(*********************************** G.D S.p.A. - Technical Department ***********************************
============= PROGRAM INFO ============
FOLDER:             TBD
MACHINES INVOLVED:  TBD 

============= DESCRIPTION =============
csp machine declaration

============= REVISIONS ===============
Date		Version	 	Author      	Description             
----------	-------		------------  	--------------------------------------------
2019/04/05 	0000.00	 	M.Grasso		Creation of the PRG

**********************************************************************************************************)
(*$R process_ref := prc; $*)
PROGRAM csp_case_feed_shuttle
VAR
	
	prc:											process;
	prc_path:										STRING;
	
END_VAR

_read_var_input();

_object_manager();

IF 	NOT objects_running()
THEN
	RETURN;	
END_IF

_read_process_image();

_mode_manager();

CASE process_get_mode(prc) OF
	MODE_ABSENT,
	MODE_INACTIVE:
		RETURN;
	MODE_TEST:
		_handle_process_test();
END_CASE

_set_runtime_properties();

(********************************* BODY *********************************)
(************************************************************************)

_handle_messages();

_write_output();

ACTION _handle_messages:
;
END_ACTION

ACTION _handle_process_test:
;
END_ACTION

ACTION _mode_manager:
IF process_mode_req_is_pending(prc)
THEN
    process_apply_mode_req_first_step(prc);
    CASE process_get_mode(prc) OF
        MODE_TO_ABSENT:
			;
        MODE_TO_INACTIVE:
			;
        MODE_TO_TEST:
			;
        MODE_TO_OPERATIONAL:
			;
    END_CASE
    process_apply_mode_req_second_step(prc);
END_IF
END_ACTION

ACTION _object_manager:
IF objects_initialization()
THEN
	sub_process_init(
		object_name					:= 'csp_case_feed_shuttle.prc', 
		process						:= csp_case_feed.prc, 
		CONVERSION_this				:= prc);
		
	prc_path 						:= process_get_path(prc);
		
END_IF

IF objects_running()
THEN
	process_cycle(prc);
END_IF
END_ACTION

ACTION _read_process_image:
;
END_ACTION

ACTION _read_var_input:
;
END_ACTION

ACTION _set_runtime_properties:
;
END_ACTION

ACTION _write_output:
;
END_ACTION

END_PROGRAM

(* stored: Version 1.1.0.1, ProductVersion 3.1.4024.3
   POU csp_case_feed_shuttle: Id {72f32f81-a021-0d76-08c3-89e071438a4e}, SpecialFunc None
   Action _handle_messages: Id {796de86d-2e13-0899-0f8f-3af1fb469c5e}
   Action _handle_process_test: Id {18b78a19-1fe2-0a5d-244e-4acb46a14d8b}
   Action _mode_manager: Id {eca15615-6404-081e-328b-60476a479ae6}
   Action _object_manager: Id {74d7ce34-3dcb-0f77-37d4-380408d2d208}
   Action _read_process_image: Id {8fe2780c-3908-0ad8-03c0-64c80177a22f}
   Action _read_var_input: Id {511cd5cb-bbf9-053f-3cf2-3dc434928c62}
   Action _set_runtime_properties: Id {e0222b58-bc14-031b-0fa0-534941d6bae2}
   Action _write_output: Id {572edf53-719b-0d5e-0010-60c65fb86ccf} *)
